# EPICS autosave request: NDFileIMMApp/Db/NDFileIMM_settings.req
file "NDPluginFile_settings.req", P=$(P), R=$(R)
$(P)$(R)FilePath
$(P)$(R)FileName
$(P)$(R)FileNumber
$(P)$(R)AutoIncrement
$(P)$(R)FileTemplate
$(P)$(R)AutoSave
$(P)$(R)FileFormat
$(P)$(R)FileWriteMode
$(P)$(R)NumCapture
$(P)$(R)EnableCallbacks
$(P)$(R)NDFileIMM_throw_images
$(P)$(R)NDAttributesFile
